FUNCTION_BLOCK EL3318
VAR
	_io : EL3xx8_Data;
	{attribute addProperty Name "WcState"}
	_wcState : WcStateInputToggle;
	{attribute addProperty Name "Info data"}
	_infoData : InfoDataAds;
END_VAR

PROPERTY IO : REFERENCE TO EL3xx8_Data
GET
IO REF= _io;
END_GET
END_PROPERTY

PROPERTY WcState : REFERENCE TO WcStateInputToggle
GET
WcState REF= _wcState;
END_GET
END_PROPERTY

END_FUNCTION_BLOCK

(* stored: Version 1.1.0.1, ProductVersion 3.1.4024.9
   POU EL3318: Id {7bb7ada6-0c1c-08f4-3eef-0d097c8b2365}, SpecialFunc None
   Property IO: Id {c834b1cb-48cd-0489-23dd-ed58fed23d0c}
   Get Get: Id {6f9ee7ec-a136-0714-151a-52280313779d}
   Property WcState: Id {29d1067d-fb9f-02f0-37d9-e71a95215ca8}
   Get Get: Id {13554685-c4a2-0773-1c5d-8f4a239a87a1} *)
